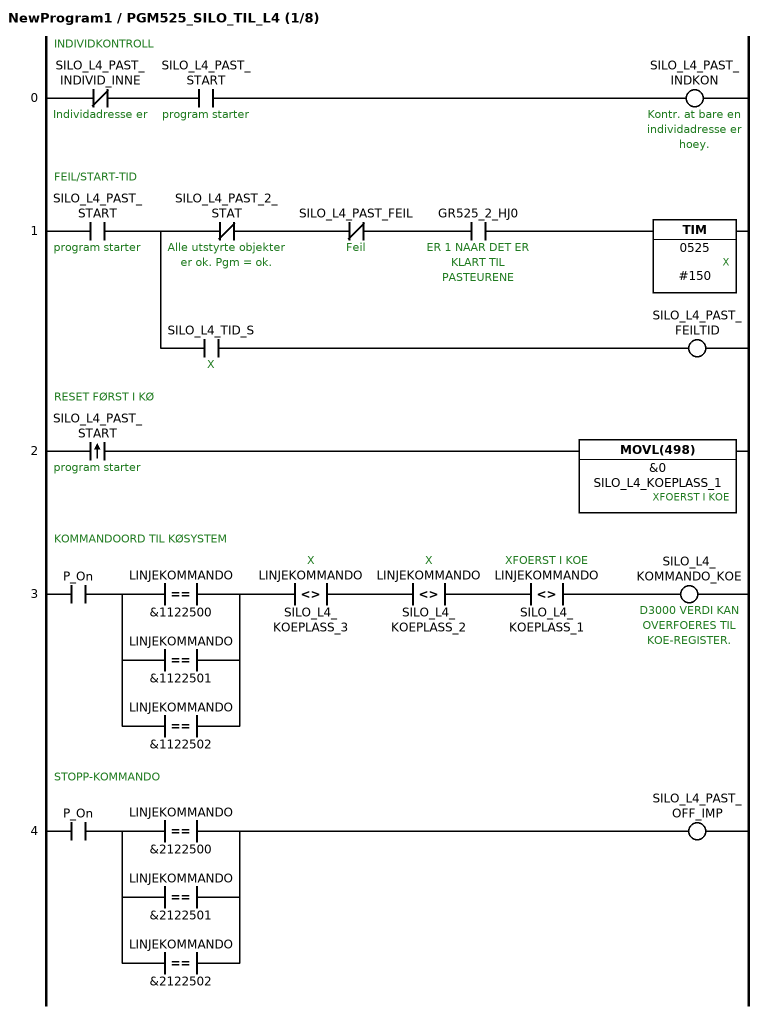
; [picture p672: NewProgram1 / PGM525_SILO_TIL_L4, rungs 0-4]
; rung 0: INDIVIDKONTROLL
LDNOT SILO_L4_PAST_INDIVID_INNE  ; Individadresse er
AND SILO_L4_PAST_START  ; program starter
OUT SILO_L4_PAST_INDKON  ; Kontr. at bare en individadresse er hoey.
; rung 1: FEIL/START-TID
LD SILO_L4_PAST_START  ; program starter
OUT TR0
ANDNOT SILO_L4_PAST_2_STAT  ; Alle utstyrte objekter er ok. Pgm = ok.
ANDNOT SILO_L4_PAST_FEIL  ; Feil
AND GR525_2_HJ0  ; ER 1 NAAR DET ER KLART TIL PASTEURENE
TIM 0525 #150  ; X
LD TR0
AND SILO_L4_TID_S  ; X
OUT SILO_L4_PAST_FEILTID
; rung 2: RESET FØRST I KØ
@LD SILO_L4_PAST_START  ; program starter
MOVL(498) &0 SILO_L4_KOEPLASS_1  ; XFOERST I KOE
; rung 3: KOMMANDOORD TIL KØSYSTEM
LD P_On
LD=L(301) LINJEKOMMANDO &1122500
OR=L(301) LINJEKOMMANDO &1122501
OR=L(301) LINJEKOMMANDO &1122502
ANDLD
AND<>L(306) LINJEKOMMANDO SILO_L4_KOEPLASS_3  ; X
AND<>L(306) LINJEKOMMANDO SILO_L4_KOEPLASS_2  ; X
AND<>L(306) LINJEKOMMANDO SILO_L4_KOEPLASS_1  ; XFOERST I KOE
OUT SILO_L4_KOMMANDO_KOE  ; D3000 VERDI KAN OVERFOERES TIL KOE-REGISTER.
; rung 4: STOPP-KOMMANDO
LD P_On
LD=L(301) LINJEKOMMANDO &2122500
OR=L(301) LINJEKOMMANDO &2122501
OR=L(301) LINJEKOMMANDO &2122502
ANDLD
OUT SILO_L4_PAST_OFF_IMP

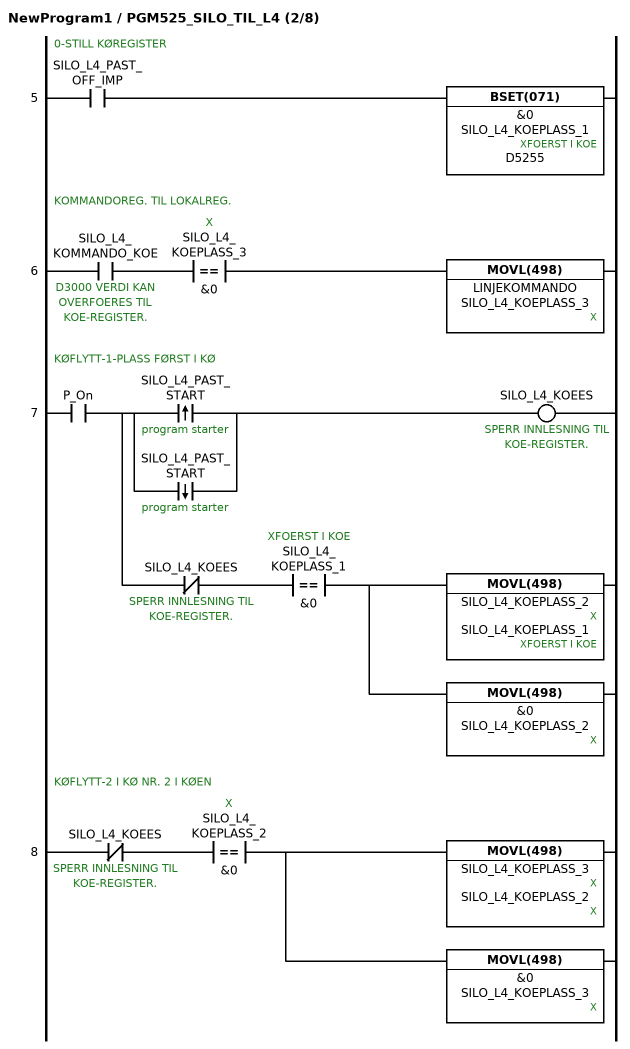
; rung 5: 0-STILL KØREGISTER
LD SILO_L4_PAST_OFF_IMP
BSET(071) &0 SILO_L4_KOEPLASS_1 D5255  ; XFOERST I KOE
; rung 6: KOMMANDOREG. TIL LOKALREG.
LD SILO_L4_KOMMANDO_KOE  ; D3000 VERDI KAN OVERFOERES TIL KOE-REGISTER.
AND=L(301) SILO_L4_KOEPLASS_3 &0  ; X
MOVL(498) LINJEKOMMANDO SILO_L4_KOEPLASS_3  ; X
; rung 7: KØFLYTT-1-PLASS FØRST I KØ
LD P_On
OUT TR0
@LD SILO_L4_PAST_START  ; program starter
%OR SILO_L4_PAST_START  ; program starter
ANDLD
OUT SILO_L4_KOEES  ; SPERR INNLESNING TIL KOE-REGISTER.
LD TR0
ANDNOT SILO_L4_KOEES  ; SPERR INNLESNING TIL KOE-REGISTER.
AND=L(301) SILO_L4_KOEPLASS_1 &0  ; XFOERST I KOE
MOVL(498) SILO_L4_KOEPLASS_2 SILO_L4_KOEPLASS_1  ; X, XFOERST I KOE
MOVL(498) &0 SILO_L4_KOEPLASS_2  ; X
; rung 8: KØFLYTT-2 I KØ NR. 2 I KØEN
LDNOT SILO_L4_KOEES  ; SPERR INNLESNING TIL KOE-REGISTER.
AND=L(301) SILO_L4_KOEPLASS_2 &0  ; X
MOVL(498) SILO_L4_KOEPLASS_3 SILO_L4_KOEPLASS_2  ; X
MOVL(498) &0 SILO_L4_KOEPLASS_3  ; X

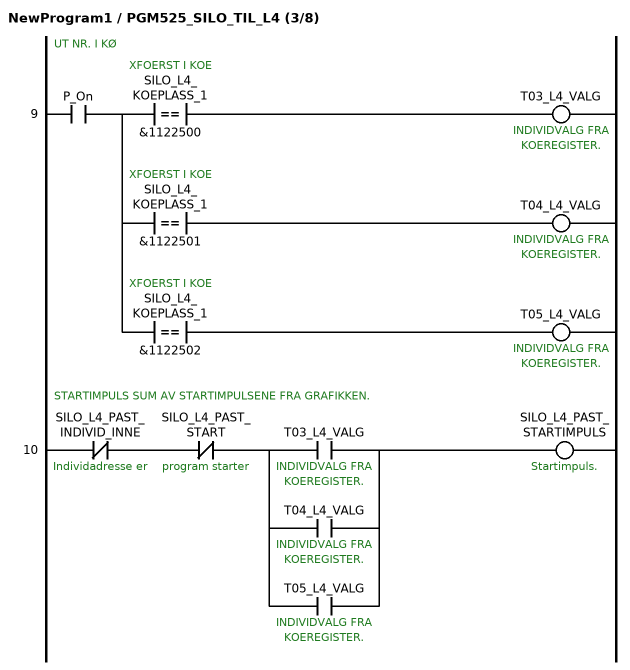
; rung 9: UT NR. I KØ
LD P_On
OUT TR0
AND=L(301) SILO_L4_KOEPLASS_1 &1122500  ; XFOERST I KOE
OUT T03_L4_VALG  ; INDIVIDVALG FRA KOEREGISTER.
LD TR0
AND=L(301) SILO_L4_KOEPLASS_1 &1122501  ; XFOERST I KOE
OUT T04_L4_VALG  ; INDIVIDVALG FRA KOEREGISTER.
LD TR0
AND=L(301) SILO_L4_KOEPLASS_1 &1122502  ; XFOERST I KOE
OUT T05_L4_VALG  ; INDIVIDVALG FRA KOEREGISTER.
; rung 10: STARTIMPULS SUM AV STARTIMPULSENE FRA GRAFIKKEN.
LDNOT SILO_L4_PAST_INDIVID_INNE  ; Individadresse er
ANDNOT SILO_L4_PAST_START  ; program starter
LD T03_L4_VALG  ; INDIVIDVALG FRA KOEREGISTER.
OR T04_L4_VALG  ; INDIVIDVALG FRA KOEREGISTER.
OR T05_L4_VALG  ; INDIVIDVALG FRA KOEREGISTER.
ANDLD
OUT SILO_L4_PAST_STARTIMPULS  ; Startimpuls.

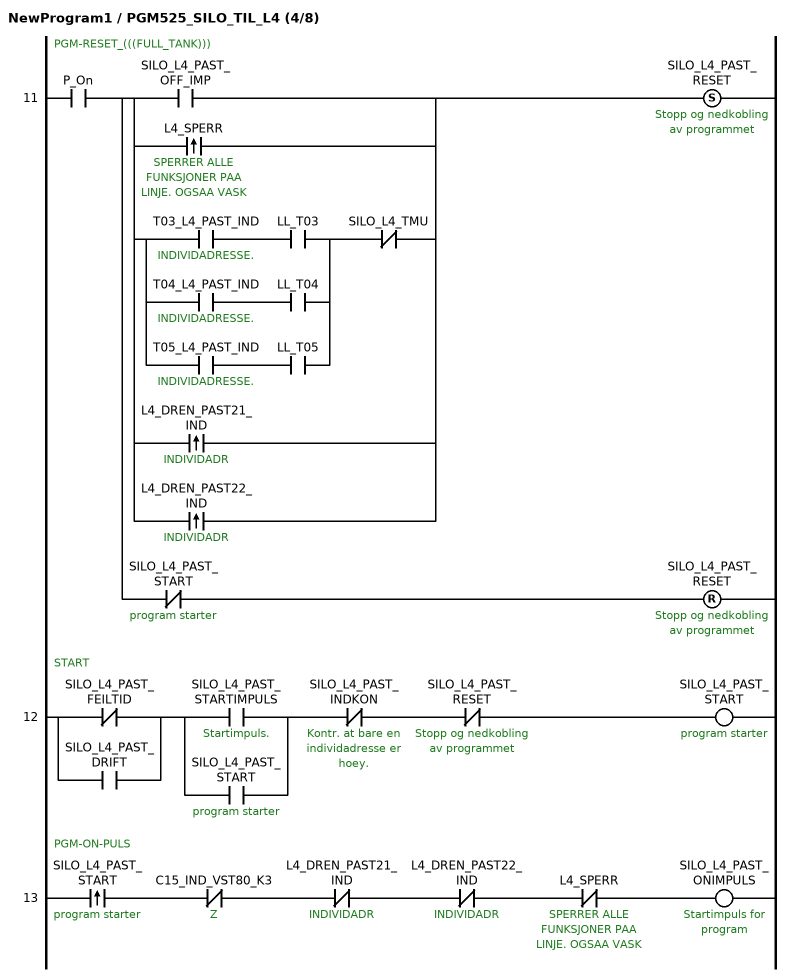
; rung 11: PGM-RESET_(((FULL_TANK)))
LD P_On
OUT TR0
LD SILO_L4_PAST_OFF_IMP
@OR L4_SPERR  ; SPERRER ALLE FUNKSJONER PAA LINJE. OGSAA VASK
LD T03_L4_PAST_IND  ; INDIVIDADRESSE.
AND LL_T03
LD T04_L4_PAST_IND  ; INDIVIDADRESSE.
AND LL_T04
ORLD
LD T05_L4_PAST_IND  ; INDIVIDADRESSE.
AND LL_T05
ORLD
ANDNOT SILO_L4_TMU
ORLD
@OR L4_DREN_PAST21_IND  ; INDIVIDADR
@OR L4_DREN_PAST22_IND  ; INDIVIDADR
ANDLD
SET SILO_L4_PAST_RESET  ; Stopp og nedkobling av programmet
LD TR0
ANDNOT SILO_L4_PAST_START  ; program starter
RSET SILO_L4_PAST_RESET  ; Stopp og nedkobling av programmet
; rung 12: START
LDNOT SILO_L4_PAST_FEILTID
OR SILO_L4_PAST_DRIFT
LD SILO_L4_PAST_STARTIMPULS  ; Startimpuls.
OR SILO_L4_PAST_START  ; program starter
ANDLD
ANDNOT SILO_L4_PAST_INDKON  ; Kontr. at bare en individadresse er hoey.
ANDNOT SILO_L4_PAST_RESET  ; Stopp og nedkobling av programmet
OUT SILO_L4_PAST_START  ; program starter
; rung 13: PGM-ON-PULS
@LD SILO_L4_PAST_START  ; program starter
ANDNOT C15_IND_VST80_K3  ; Z
ANDNOT L4_DREN_PAST21_IND  ; INDIVIDADR
ANDNOT L4_DREN_PAST22_IND  ; INDIVIDADR
ANDNOT L4_SPERR  ; SPERRER ALLE FUNKSJONER PAA LINJE. OGSAA VASK
OUT SILO_L4_PAST_ONIMPULS  ; Startimpuls for  program

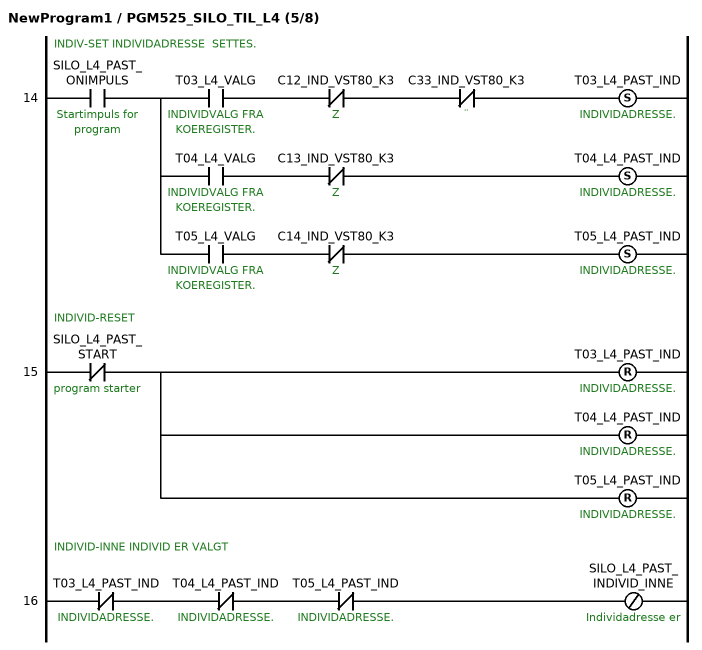
; rung 14: INDIV-SET INDIVIDADRESSE  SETTES.
LD SILO_L4_PAST_ONIMPULS  ; Startimpuls for  program
OUT TR0
AND T03_L4_VALG  ; INDIVIDVALG FRA KOEREGISTER.
ANDNOT C12_IND_VST80_K3  ; Z
ANDNOT C33_IND_VST80_K3  ; ¨
SET T03_L4_PAST_IND  ; INDIVIDADRESSE.
LD TR0
AND T04_L4_VALG  ; INDIVIDVALG FRA KOEREGISTER.
ANDNOT C13_IND_VST80_K3  ; Z
SET T04_L4_PAST_IND  ; INDIVIDADRESSE.
LD TR0
AND T05_L4_VALG  ; INDIVIDVALG FRA KOEREGISTER.
ANDNOT C14_IND_VST80_K3  ; Z
SET T05_L4_PAST_IND  ; INDIVIDADRESSE.
; rung 15: INDIVID-RESET
LDNOT SILO_L4_PAST_START  ; program starter
RSET T03_L4_PAST_IND  ; INDIVIDADRESSE.
RSET T04_L4_PAST_IND  ; INDIVIDADRESSE.
RSET T05_L4_PAST_IND  ; INDIVIDADRESSE.
; rung 16: INDIVID-INNE INDIVID ER VALGT
LDNOT T03_L4_PAST_IND  ; INDIVIDADRESSE.
ANDNOT T04_L4_PAST_IND  ; INDIVIDADRESSE.
ANDNOT T05_L4_PAST_IND  ; INDIVIDADRESSE.
OUTNOT SILO_L4_PAST_INDIVID_INNE  ; Individadresse er

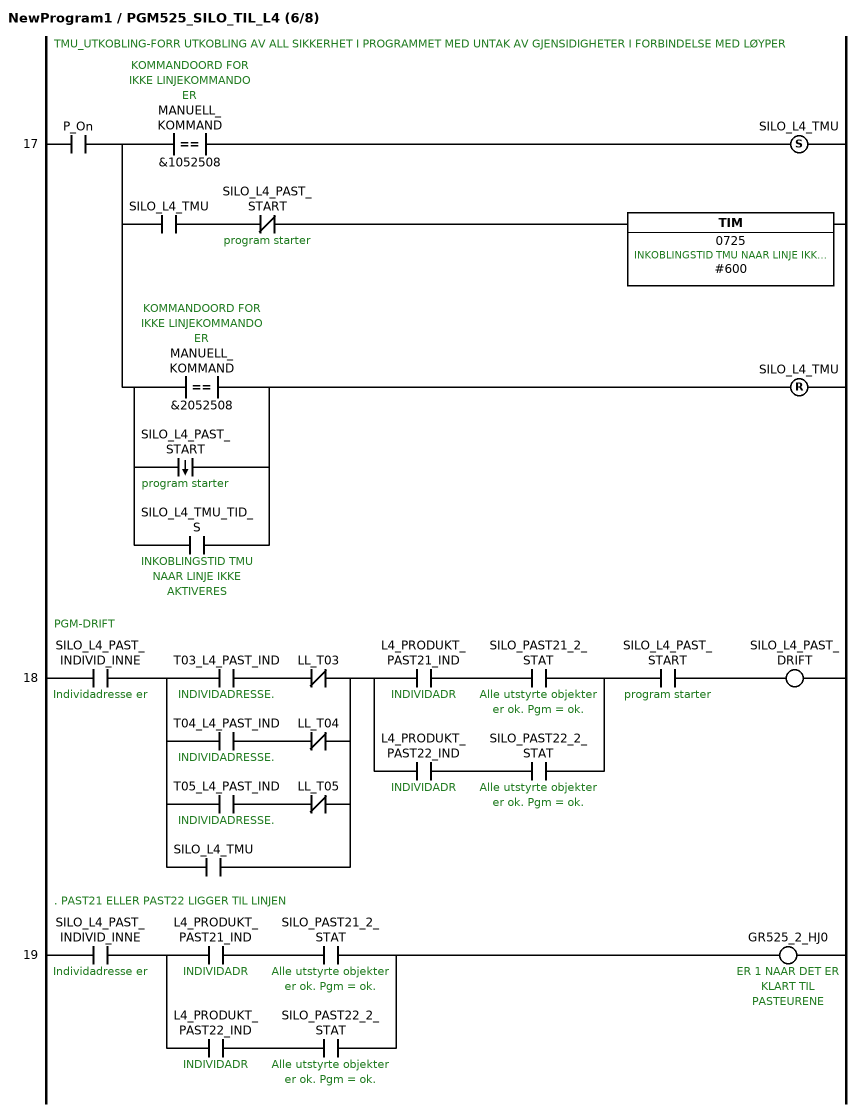
; rung 17: TMU_UTKOBLING-FORR UTKOBLING AV ALL SIKKERHET I PROGRAMMET MED UNTAK AV GJENSIDIGHETER I FORBINDELSE MED LØYPER
LD P_On
OUT TR0
AND=L(301) MANUELL_KOMMAND &1052508  ; KOMMANDOORD FOR IKKE LINJEKOMMANDOER
SET SILO_L4_TMU
LD TR0
AND SILO_L4_TMU
ANDNOT SILO_L4_PAST_START  ; program starter
TIM 0725 #600  ; INKOBLINGSTID TMU NAAR LINJE IKKE AKTIVERES
LD TR0
LD=L(301) MANUELL_KOMMAND &2052508  ; KOMMANDOORD FOR IKKE LINJEKOMMANDOER
%OR SILO_L4_PAST_START  ; program starter
OR SILO_L4_TMU_TID_S  ; INKOBLINGSTID TMU NAAR LINJE IKKE AKTIVERES
ANDLD
RSET SILO_L4_TMU
; rung 18: PGM-DRIFT
LD SILO_L4_PAST_INDIVID_INNE  ; Individadresse er
LD T03_L4_PAST_IND  ; INDIVIDADRESSE.
ANDNOT LL_T03
LD T04_L4_PAST_IND  ; INDIVIDADRESSE.
ANDNOT LL_T04
ORLD
LD T05_L4_PAST_IND  ; INDIVIDADRESSE.
ANDNOT LL_T05
ORLD
OR SILO_L4_TMU
ANDLD
LD L4_PRODUKT_PAST21_IND  ; INDIVIDADR
AND SILO_PAST21_2_STAT  ; Alle utstyrte objekter er ok. Pgm = ok.
LD L4_PRODUKT_PAST22_IND  ; INDIVIDADR
AND SILO_PAST22_2_STAT  ; Alle utstyrte objekter er ok. Pgm = ok.
ORLD
ANDLD
AND SILO_L4_PAST_START  ; program starter
OUT SILO_L4_PAST_DRIFT
; rung 19: . PAST21 ELLER PAST22 LIGGER TIL LINJEN
LD SILO_L4_PAST_INDIVID_INNE  ; Individadresse er
LD L4_PRODUKT_PAST21_IND  ; INDIVIDADR
AND SILO_PAST21_2_STAT  ; Alle utstyrte objekter er ok. Pgm = ok.
LD L4_PRODUKT_PAST22_IND  ; INDIVIDADR
AND SILO_PAST22_2_STAT  ; Alle utstyrte objekter er ok. Pgm = ok.
ORLD
ANDLD
OUT GR525_2_HJ0  ; ER 1 NAAR DET ER KLART TIL PASTEURENE

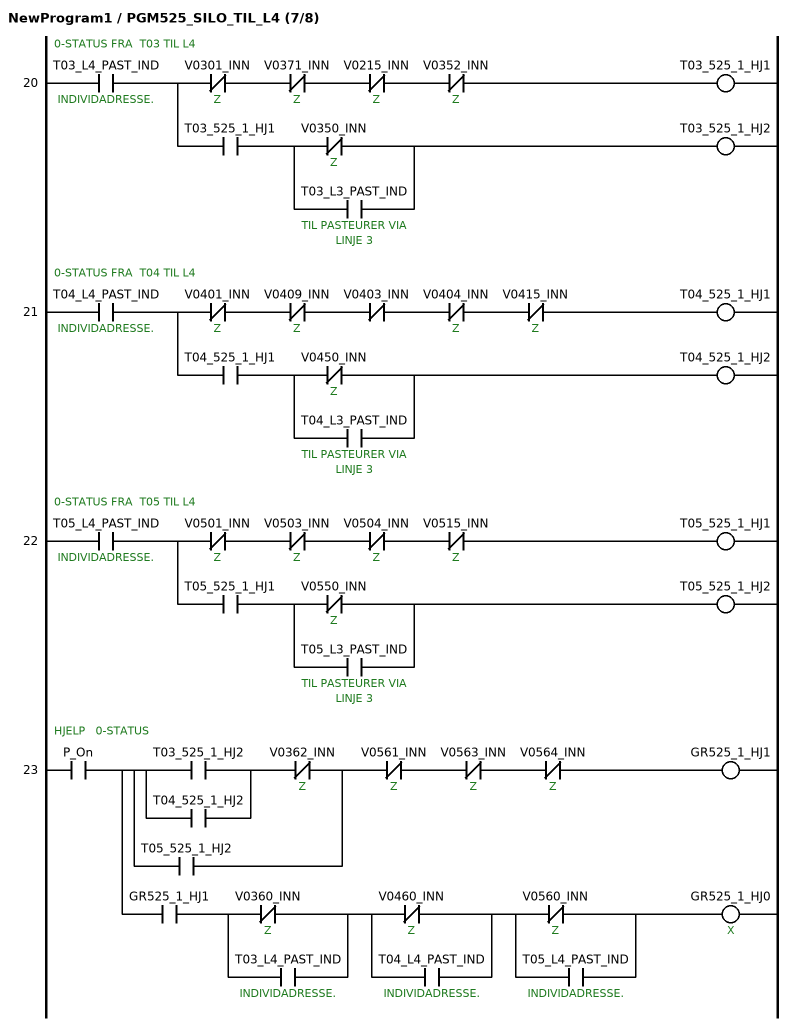
; rung 20: 0-STATUS FRA  T03 TIL L4
LD T03_L4_PAST_IND  ; INDIVIDADRESSE.
OUT TR0
ANDNOT V0301_INN  ; Z
ANDNOT V0371_INN  ; Z
ANDNOT V0215_INN  ; Z
ANDNOT V0352_INN  ; Z
OUT T03_525_1_HJ1
LD TR0
AND T03_525_1_HJ1
LDNOT V0350_INN  ; Z
OR T03_L3_PAST_IND  ; TIL PASTEURER VIA LINJE 3
ANDLD
OUT T03_525_1_HJ2
; rung 21: 0-STATUS FRA  T04 TIL L4
LD T04_L4_PAST_IND  ; INDIVIDADRESSE.
OUT TR0
ANDNOT V0401_INN  ; Z
ANDNOT V0409_INN  ; Z
ANDNOT V0403_INN
ANDNOT V0404_INN  ; Z
ANDNOT V0415_INN  ; Z
OUT T04_525_1_HJ1
LD TR0
AND T04_525_1_HJ1
LDNOT V0450_INN  ; Z
OR T04_L3_PAST_IND  ; TIL PASTEURER VIA LINJE 3
ANDLD
OUT T04_525_1_HJ2
; rung 22: 0-STATUS FRA  T05 TIL L4
LD T05_L4_PAST_IND  ; INDIVIDADRESSE.
OUT TR0
ANDNOT V0501_INN  ; Z
ANDNOT V0503_INN  ; Z
ANDNOT V0504_INN  ; Z
ANDNOT V0515_INN  ; Z
OUT T05_525_1_HJ1
LD TR0
AND T05_525_1_HJ1
LDNOT V0550_INN  ; Z
OR T05_L3_PAST_IND  ; TIL PASTEURER VIA LINJE 3
ANDLD
OUT T05_525_1_HJ2
; rung 23: HJELP   0-STATUS
LD P_On
OUT TR0
LD T03_525_1_HJ2
OR T04_525_1_HJ2
ANDNOT V0362_INN  ; Z
OR T05_525_1_HJ2
ANDLD
ANDNOT V0561_INN  ; Z
ANDNOT V0563_INN  ; Z
ANDNOT V0564_INN  ; Z
OUT GR525_1_HJ1
LD TR0
AND GR525_1_HJ1
LDNOT V0360_INN  ; Z
OR T03_L4_PAST_IND  ; INDIVIDADRESSE.
ANDLD
LDNOT V0460_INN  ; Z
OR T04_L4_PAST_IND  ; INDIVIDADRESSE.
ANDLD
LDNOT V0560_INN  ; Z
OR T05_L4_PAST_IND  ; INDIVIDADRESSE.
ANDLD
OUT GR525_1_HJ0  ; X

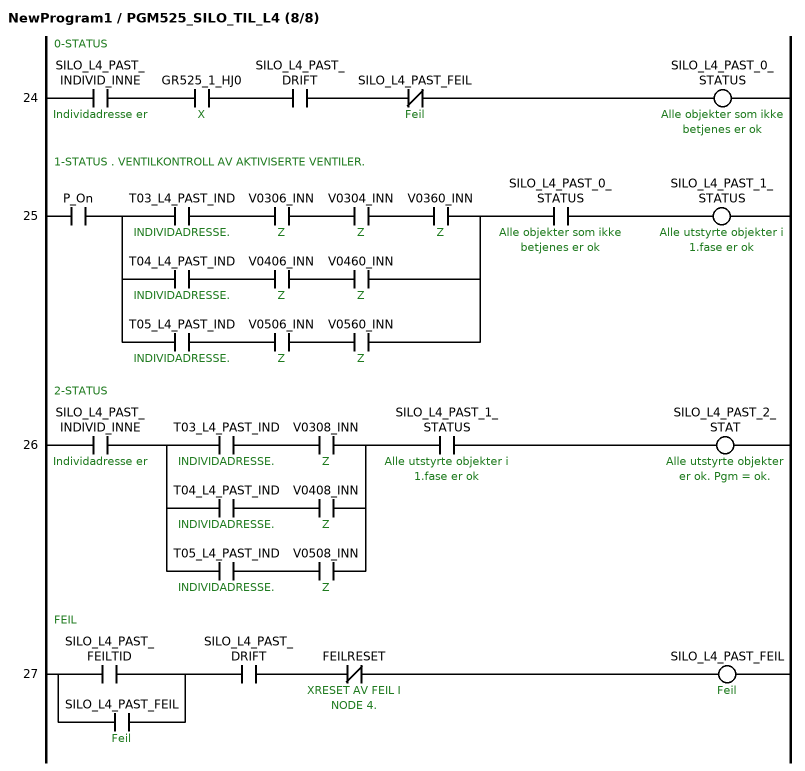
; rung 24: 0-STATUS
LD SILO_L4_PAST_INDIVID_INNE  ; Individadresse er
AND GR525_1_HJ0  ; X
AND SILO_L4_PAST_DRIFT
ANDNOT SILO_L4_PAST_FEIL  ; Feil
OUT SILO_L4_PAST_0_STATUS  ; Alle objekter som ikke betjenes er ok
; rung 25: 1-STATUS . VENTILKONTROLL AV AKTIVISERTE VENTILER.
LD P_On
LD T03_L4_PAST_IND  ; INDIVIDADRESSE.
AND V0306_INN  ; Z
AND V0304_INN  ; Z
AND V0360_INN  ; Z
LD T04_L4_PAST_IND  ; INDIVIDADRESSE.
AND V0406_INN  ; Z
AND V0460_INN  ; Z
ORLD
LD T05_L4_PAST_IND  ; INDIVIDADRESSE.
AND V0506_INN  ; Z
AND V0560_INN  ; Z
ORLD
ANDLD
AND SILO_L4_PAST_0_STATUS  ; Alle objekter som ikke betjenes er ok
OUT SILO_L4_PAST_1_STATUS  ; Alle utstyrte objekter i 1.fase er ok
; rung 26: 2-STATUS
LD SILO_L4_PAST_INDIVID_INNE  ; Individadresse er
LD T03_L4_PAST_IND  ; INDIVIDADRESSE.
AND V0308_INN  ; Z
LD T04_L4_PAST_IND  ; INDIVIDADRESSE.
AND V0408_INN  ; Z
ORLD
LD T05_L4_PAST_IND  ; INDIVIDADRESSE.
AND V0508_INN  ; Z
ORLD
ANDLD
AND SILO_L4_PAST_1_STATUS  ; Alle utstyrte objekter i 1.fase er ok
OUT SILO_L4_PAST_2_STAT  ; Alle utstyrte objekter er ok. Pgm = ok.
; rung 27: FEIL
LD SILO_L4_PAST_FEILTID
OR SILO_L4_PAST_FEIL  ; Feil
AND SILO_L4_PAST_DRIFT
ANDNOT FEILRESET  ; XRESET AV FEIL I NODE 4.
OUT SILO_L4_PAST_FEIL  ; Feil

### Section PGM526_TIL_PAST21

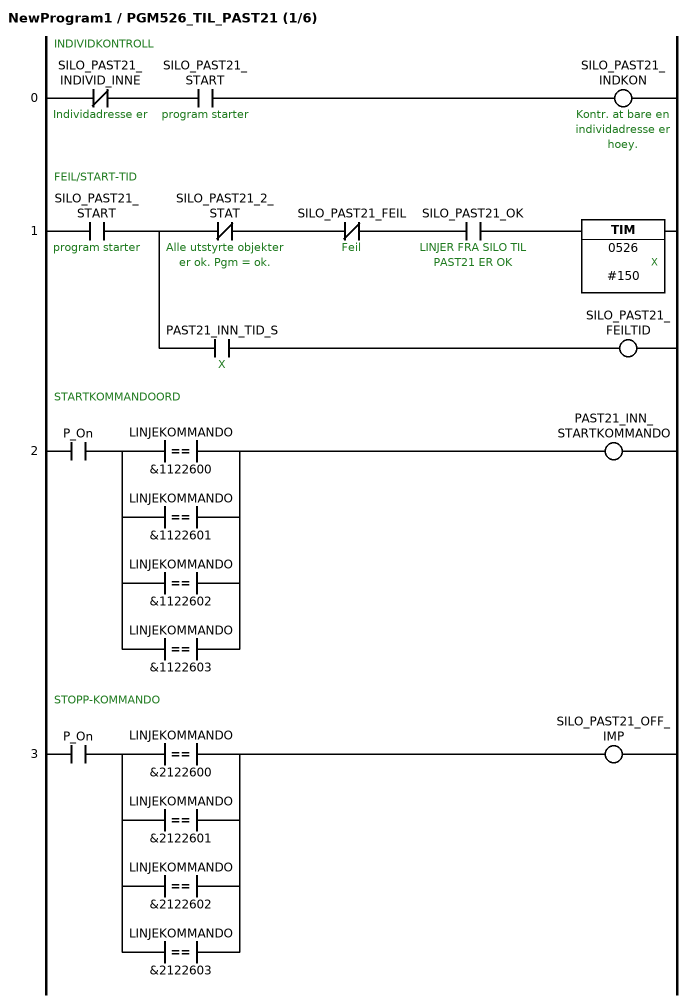
; rung 0: INDIVIDKONTROLL
LDNOT SILO_PAST21_INDIVID_INNE  ; Individadresse er
AND SILO_PAST21_START  ; program starter
OUT SILO_PAST21_INDKON  ; Kontr. at bare en individadresse er hoey.
; rung 1: FEIL/START-TID
LD SILO_PAST21_START  ; program starter
OUT TR0
ANDNOT SILO_PAST21_2_STAT  ; Alle utstyrte objekter er ok. Pgm = ok.
ANDNOT SILO_PAST21_FEIL  ; Feil
AND SILO_PAST21_OK  ; LINJER FRA SILO TIL  PAST21 ER OK
TIM 0526 #150  ; X
LD TR0
AND PAST21_INN_TID_S  ; X
OUT SILO_PAST21_FEILTID
; rung 2: STARTKOMMANDOORD
LD P_On
LD=L(301) LINJEKOMMANDO &1122600
OR=L(301) LINJEKOMMANDO &1122601
OR=L(301) LINJEKOMMANDO &1122602
OR=L(301) LINJEKOMMANDO &1122603
ANDLD
OUT PAST21_INN_STARTKOMMANDO
; rung 3: STOPP-KOMMANDO
LD P_On
LD=L(301) LINJEKOMMANDO &2122600
OR=L(301) LINJEKOMMANDO &2122601
OR=L(301) LINJEKOMMANDO &2122602
OR=L(301) LINJEKOMMANDO &2122603
ANDLD
OUT SILO_PAST21_OFF_IMP

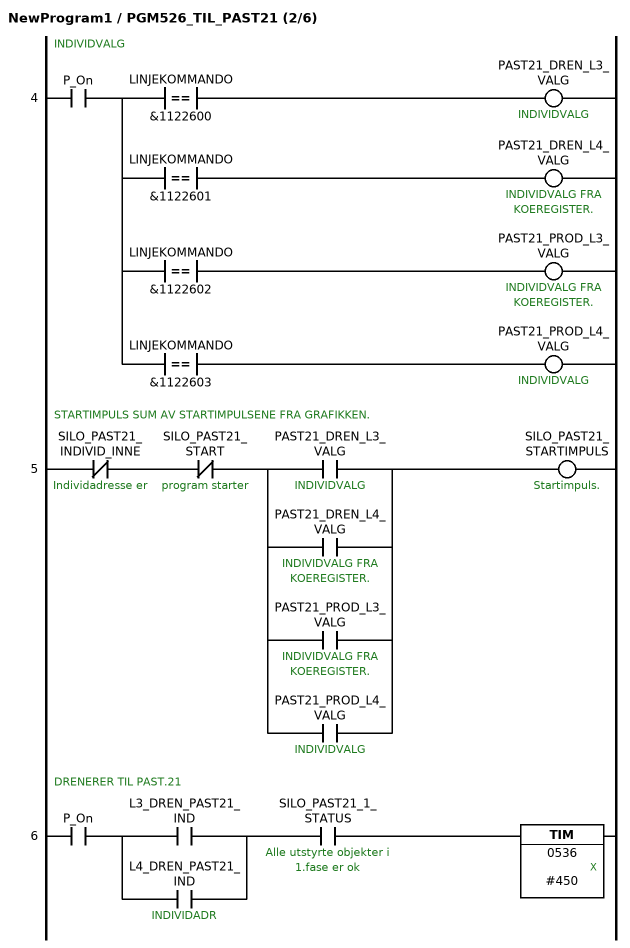
; rung 4: INDIVIDVALG
LD P_On
OUT TR0
AND=L(301) LINJEKOMMANDO &1122600
OUT PAST21_DREN_L3_VALG  ; INDIVIDVALG
LD TR0
AND=L(301) LINJEKOMMANDO &1122601
OUT PAST21_DREN_L4_VALG  ; INDIVIDVALG FRA KOEREGISTER.
LD TR0
AND=L(301) LINJEKOMMANDO &1122602
OUT PAST21_PROD_L3_VALG  ; INDIVIDVALG FRA KOEREGISTER.
LD TR0
AND=L(301) LINJEKOMMANDO &1122603
OUT PAST21_PROD_L4_VALG  ; INDIVIDVALG
; rung 5: STARTIMPULS SUM AV STARTIMPULSENE FRA GRAFIKKEN.
LDNOT SILO_PAST21_INDIVID_INNE  ; Individadresse er
ANDNOT SILO_PAST21_START  ; program starter
LD PAST21_DREN_L3_VALG  ; INDIVIDVALG
OR PAST21_DREN_L4_VALG  ; INDIVIDVALG FRA KOEREGISTER.
OR PAST21_PROD_L3_VALG  ; INDIVIDVALG FRA KOEREGISTER.
OR PAST21_PROD_L4_VALG  ; INDIVIDVALG
ANDLD
OUT SILO_PAST21_STARTIMPULS  ; Startimpuls.
; rung 6: DRENERER TIL PAST.21
LD P_On
LD L3_DREN_PAST21_IND
OR L4_DREN_PAST21_IND  ; INDIVIDADR
ANDLD
AND SILO_PAST21_1_STATUS  ; Alle utstyrte objekter i 1.fase er ok
TIM 0536 #450  ; X

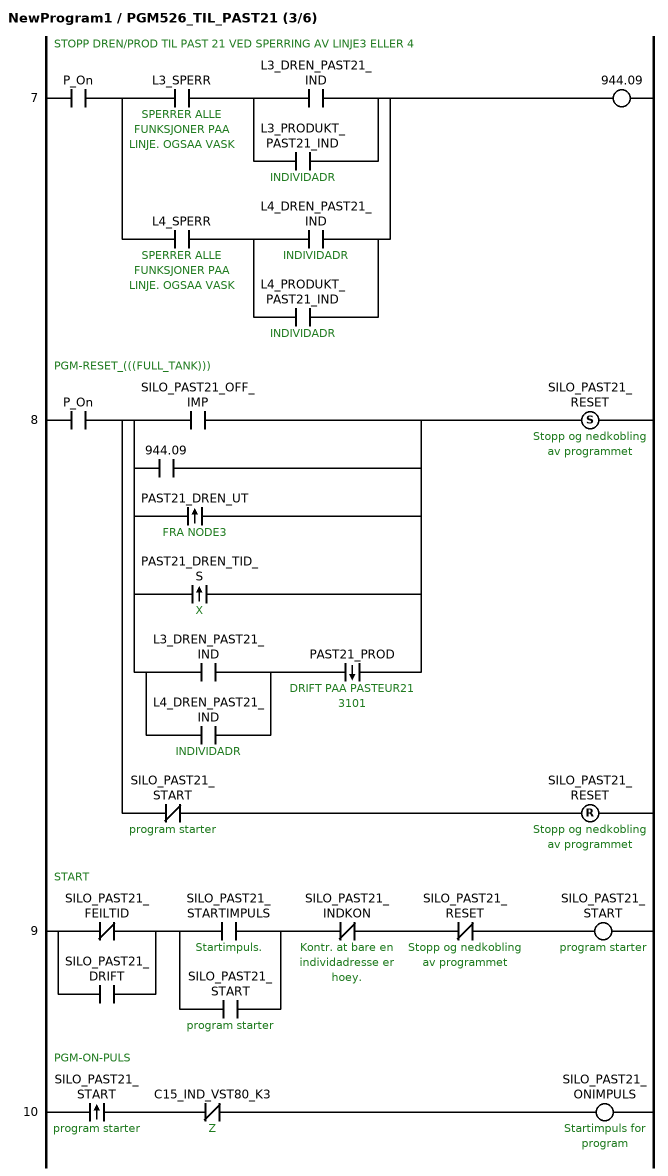
; rung 7: STOPP DREN/PROD TIL PAST 21 VED SPERRING AV LINJE3 ELLER 4
LD P_On
LD L3_SPERR  ; SPERRER ALLE FUNKSJONER PAA LINJE. OGSAA VASK
LD L3_DREN_PAST21_IND
OR L3_PRODUKT_PAST21_IND  ; INDIVIDADR
ANDLD
LD L4_SPERR  ; SPERRER ALLE FUNKSJONER PAA LINJE. OGSAA VASK
LD L4_DREN_PAST21_IND  ; INDIVIDADR
OR L4_PRODUKT_PAST21_IND  ; INDIVIDADR
ANDLD
ORLD
ANDLD
OUT 944.09
; rung 8: PGM-RESET_(((FULL_TANK)))
LD P_On
OUT TR0
LD SILO_PAST21_OFF_IMP
OR 944.09
@OR PAST21_DREN_UT  ; FRA NODE3
@OR PAST21_DREN_TID_S  ; X
LD L3_DREN_PAST21_IND
OR L4_DREN_PAST21_IND  ; INDIVIDADR
%AND PAST21_PROD  ; DRIFT PAA PASTEUR21 3101
ORLD
ANDLD
SET SILO_PAST21_RESET  ; Stopp og nedkobling av programmet
LD TR0
ANDNOT SILO_PAST21_START  ; program starter
RSET SILO_PAST21_RESET  ; Stopp og nedkobling av programmet
; rung 9: START
LDNOT SILO_PAST21_FEILTID
OR SILO_PAST21_DRIFT
LD SILO_PAST21_STARTIMPULS  ; Startimpuls.
OR SILO_PAST21_START  ; program starter
ANDLD
ANDNOT SILO_PAST21_INDKON  ; Kontr. at bare en individadresse er hoey.
ANDNOT SILO_PAST21_RESET  ; Stopp og nedkobling av programmet
OUT SILO_PAST21_START  ; program starter
; rung 10: PGM-ON-PULS
@LD SILO_PAST21_START  ; program starter
ANDNOT C15_IND_VST80_K3  ; Z
OUT SILO_PAST21_ONIMPULS  ; Startimpuls for  program

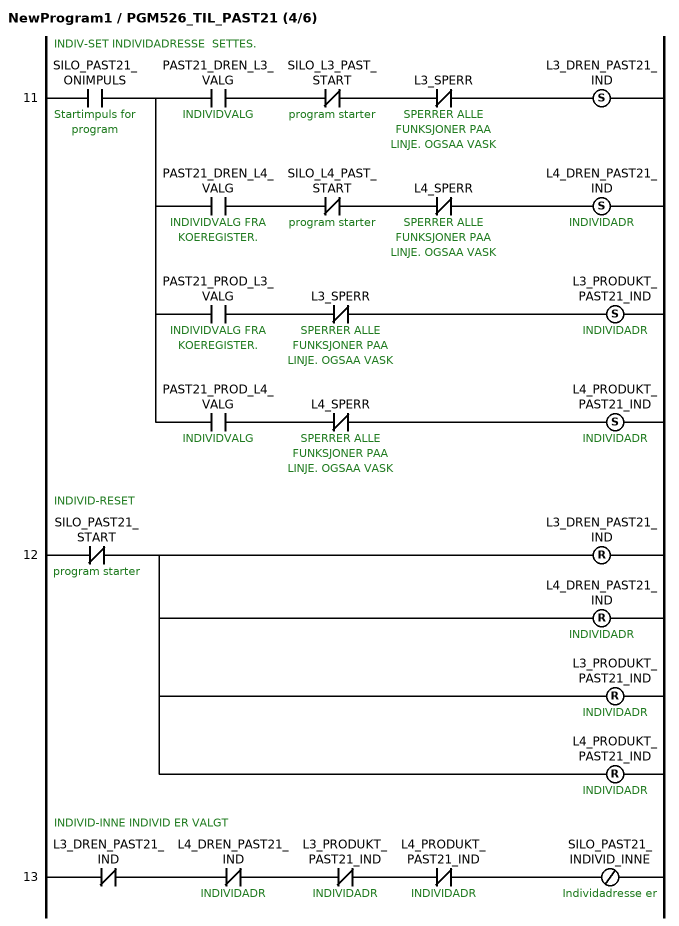
; rung 11: INDIV-SET INDIVIDADRESSE  SETTES.
LD SILO_PAST21_ONIMPULS  ; Startimpuls for  program
OUT TR0
AND PAST21_DREN_L3_VALG  ; INDIVIDVALG
ANDNOT SILO_L3_PAST_START  ; program starter
ANDNOT L3_SPERR  ; SPERRER ALLE FUNKSJONER PAA LINJE. OGSAA VASK
SET L3_DREN_PAST21_IND
LD TR0
AND PAST21_DREN_L4_VALG  ; INDIVIDVALG FRA KOEREGISTER.
ANDNOT SILO_L4_PAST_START  ; program starter
ANDNOT L4_SPERR  ; SPERRER ALLE FUNKSJONER PAA LINJE. OGSAA VASK
SET L4_DREN_PAST21_IND  ; INDIVIDADR
LD TR0
AND PAST21_PROD_L3_VALG  ; INDIVIDVALG FRA KOEREGISTER.
ANDNOT L3_SPERR  ; SPERRER ALLE FUNKSJONER PAA LINJE. OGSAA VASK
SET L3_PRODUKT_PAST21_IND  ; INDIVIDADR
LD TR0
AND PAST21_PROD_L4_VALG  ; INDIVIDVALG
ANDNOT L4_SPERR  ; SPERRER ALLE FUNKSJONER PAA LINJE. OGSAA VASK
SET L4_PRODUKT_PAST21_IND  ; INDIVIDADR
; rung 12: INDIVID-RESET
LDNOT SILO_PAST21_START  ; program starter
RSET L3_DREN_PAST21_IND
RSET L4_DREN_PAST21_IND  ; INDIVIDADR
RSET L3_PRODUKT_PAST21_IND  ; INDIVIDADR
RSET L4_PRODUKT_PAST21_IND  ; INDIVIDADR
; rung 13: INDIVID-INNE INDIVID ER VALGT
LDNOT L3_DREN_PAST21_IND
ANDNOT L4_DREN_PAST21_IND  ; INDIVIDADR
ANDNOT L3_PRODUKT_PAST21_IND  ; INDIVIDADR
ANDNOT L4_PRODUKT_PAST21_IND  ; INDIVIDADR
OUTNOT SILO_PAST21_INDIVID_INNE  ; Individadresse er

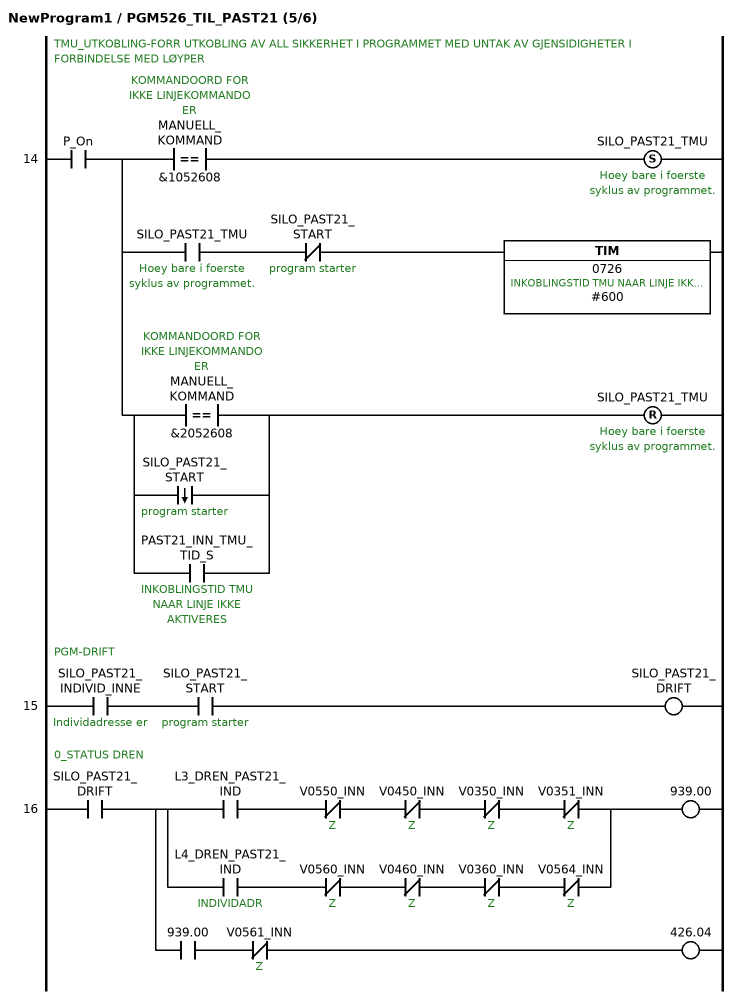
; rung 14: TMU_UTKOBLING-FORR UTKOBLING AV ALL SIKKERHET I PROGRAMMET MED UNTAK AV GJENSIDIGHETER I FORBINDELSE MED LØYPER
LD P_On
OUT TR0
AND=L(301) MANUELL_KOMMAND &1052608  ; KOMMANDOORD FOR IKKE LINJEKOMMANDOER
SET SILO_PAST21_TMU  ; Hoey bare i foerste syklus av programmet.
LD TR0
AND SILO_PAST21_TMU  ; Hoey bare i foerste syklus av programmet.
ANDNOT SILO_PAST21_START  ; program starter
TIM 0726 #600  ; INKOBLINGSTID TMU NAAR LINJE IKKE AKTIVERES
LD TR0
LD=L(301) MANUELL_KOMMAND &2052608  ; KOMMANDOORD FOR IKKE LINJEKOMMANDOER
%OR SILO_PAST21_START  ; program starter
OR PAST21_INN_TMU_TID_S  ; INKOBLINGSTID TMU NAAR LINJE IKKE AKTIVERES
ANDLD
RSET SILO_PAST21_TMU  ; Hoey bare i foerste syklus av programmet.
; rung 15: PGM-DRIFT
LD SILO_PAST21_INDIVID_INNE  ; Individadresse er
AND SILO_PAST21_START  ; program starter
OUT SILO_PAST21_DRIFT
; rung 16: 0_STATUS DREN
LD SILO_PAST21_DRIFT
OUT TR0
LD L3_DREN_PAST21_IND
ANDNOT V0550_INN  ; Z
ANDNOT V0450_INN  ; Z
ANDNOT V0350_INN  ; Z
ANDNOT V0351_INN  ; Z
LD L4_DREN_PAST21_IND  ; INDIVIDADR
ANDNOT V0560_INN  ; Z
ANDNOT V0460_INN  ; Z
ANDNOT V0360_INN  ; Z
ANDNOT V0564_INN  ; Z
ORLD
ANDLD
OUT 939.00
LD TR0
AND 939.00
ANDNOT V0561_INN  ; Z
OUT 426.04

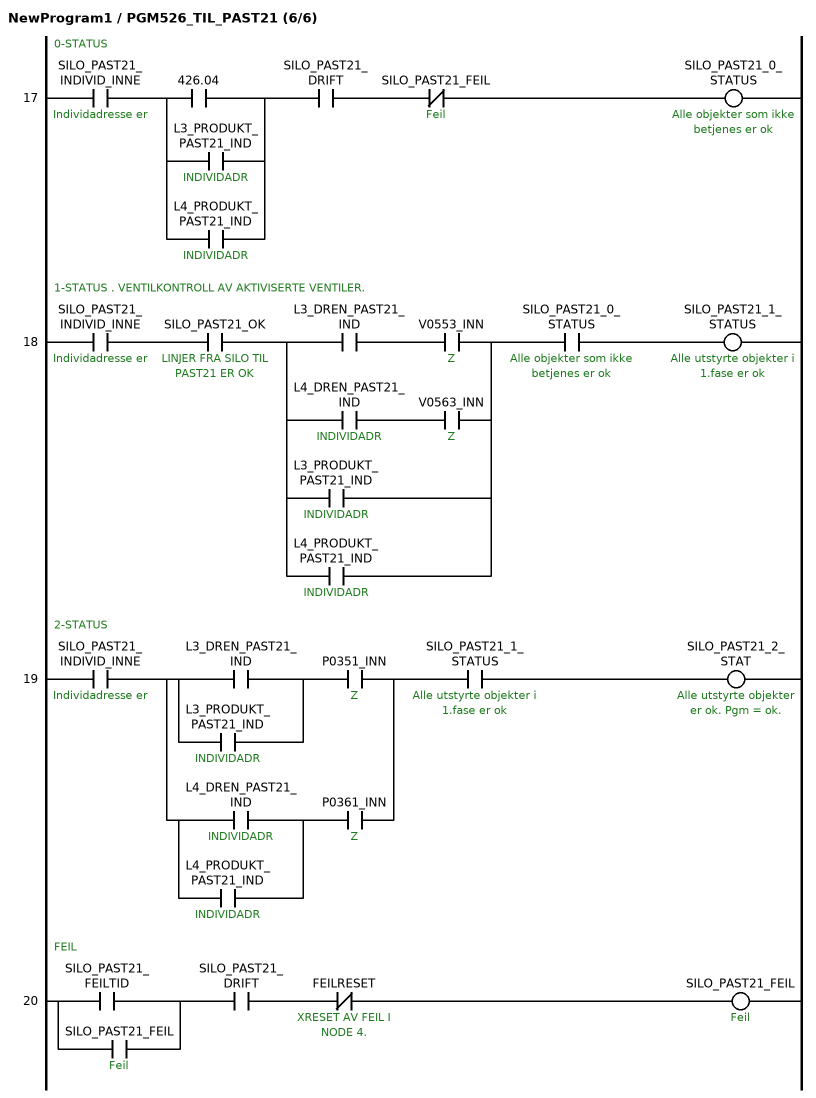
; rung 17: 0-STATUS
LD SILO_PAST21_INDIVID_INNE  ; Individadresse er
LD 426.04
OR L3_PRODUKT_PAST21_IND  ; INDIVIDADR
OR L4_PRODUKT_PAST21_IND  ; INDIVIDADR
ANDLD
AND SILO_PAST21_DRIFT
ANDNOT SILO_PAST21_FEIL  ; Feil
OUT SILO_PAST21_0_STATUS  ; Alle objekter som ikke betjenes er ok
; rung 18: 1-STATUS . VENTILKONTROLL AV AKTIVISERTE VENTILER.
LD SILO_PAST21_INDIVID_INNE  ; Individadresse er
AND SILO_PAST21_OK  ; LINJER FRA SILO TIL  PAST21 ER OK
LD L3_DREN_PAST21_IND
AND V0553_INN  ; Z
LD L4_DREN_PAST21_IND  ; INDIVIDADR
AND V0563_INN  ; Z
ORLD
OR L3_PRODUKT_PAST21_IND  ; INDIVIDADR
OR L4_PRODUKT_PAST21_IND  ; INDIVIDADR
ANDLD
AND SILO_PAST21_0_STATUS  ; Alle objekter som ikke betjenes er ok
OUT SILO_PAST21_1_STATUS  ; Alle utstyrte objekter i 1.fase er ok
; rung 19: 2-STATUS
LD SILO_PAST21_INDIVID_INNE  ; Individadresse er
LD L3_DREN_PAST21_IND
OR L3_PRODUKT_PAST21_IND  ; INDIVIDADR
AND P0351_INN  ; Z
LD L4_DREN_PAST21_IND  ; INDIVIDADR
OR L4_PRODUKT_PAST21_IND  ; INDIVIDADR
AND P0361_INN  ; Z
ORLD
ANDLD
AND SILO_PAST21_1_STATUS  ; Alle utstyrte objekter i 1.fase er ok
OUT SILO_PAST21_2_STAT  ; Alle utstyrte objekter er ok. Pgm = ok.
; rung 20: FEIL
LD SILO_PAST21_FEILTID
OR SILO_PAST21_FEIL  ; Feil
AND SILO_PAST21_DRIFT
ANDNOT FEILRESET  ; XRESET AV FEIL I NODE 4.
OUT SILO_PAST21_FEIL  ; Feil

### Section L3_STATUS

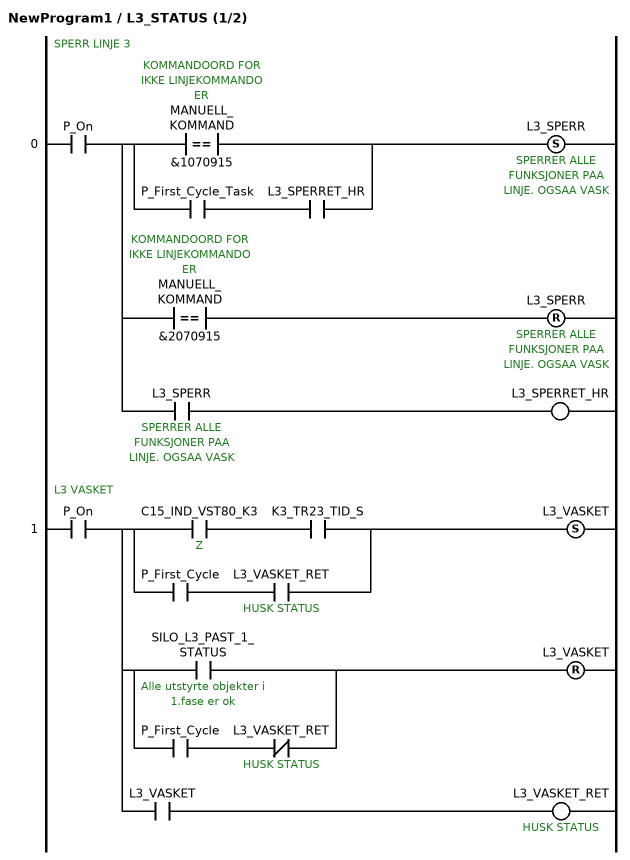
; rung 0: SPERR LINJE 3
LD P_On
OUT TR0
LD=L(301) MANUELL_KOMMAND &1070915  ; KOMMANDOORD FOR IKKE LINJEKOMMANDOER
LD P_First_Cycle_Task
AND L3_SPERRET_HR
ORLD
ANDLD
SET L3_SPERR  ; SPERRER ALLE FUNKSJONER PAA LINJE. OGSAA VASK
LD TR0
AND=L(301) MANUELL_KOMMAND &2070915  ; KOMMANDOORD FOR IKKE LINJEKOMMANDOER
RSET L3_SPERR  ; SPERRER ALLE FUNKSJONER PAA LINJE. OGSAA VASK
LD TR0
AND L3_SPERR  ; SPERRER ALLE FUNKSJONER PAA LINJE. OGSAA VASK
OUT L3_SPERRET_HR
; rung 1: L3 VASKET
LD P_On
OUT TR0
LD C15_IND_VST80_K3  ; Z
AND K3_TR23_TID_S
LD P_First_Cycle
AND L3_VASKET_RET  ; HUSK STATUS
ORLD
ANDLD
SET L3_VASKET
LD TR0
LD SILO_L3_PAST_1_STATUS  ; Alle utstyrte objekter i 1.fase er ok
LD P_First_Cycle
ANDNOT L3_VASKET_RET  ; HUSK STATUS
ORLD
ANDLD
RSET L3_VASKET
LD TR0
AND L3_VASKET
OUT L3_VASKET_RET  ; HUSK STATUS

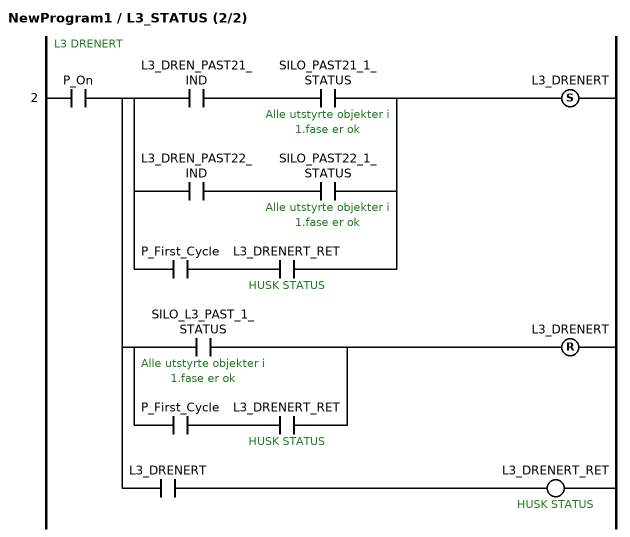
; rung 2: L3 DRENERT
LD P_On
OUT TR0
LD L3_DREN_PAST21_IND
AND SILO_PAST21_1_STATUS  ; Alle utstyrte objekter i 1.fase er ok
LD L3_DREN_PAST22_IND
AND SILO_PAST22_1_STATUS  ; Alle utstyrte objekter i 1.fase er ok
ORLD
LD P_First_Cycle
AND L3_DRENERT_RET  ; HUSK STATUS
ORLD
ANDLD
SET L3_DRENERT
LD TR0
LD SILO_L3_PAST_1_STATUS  ; Alle utstyrte objekter i 1.fase er ok
LD P_First_Cycle
AND L3_DRENERT_RET  ; HUSK STATUS
ORLD
ANDLD
RSET L3_DRENERT
LD TR0
AND L3_DRENERT
OUT L3_DRENERT_RET  ; HUSK STATUS

### Section PGM527_TIL_PAST22

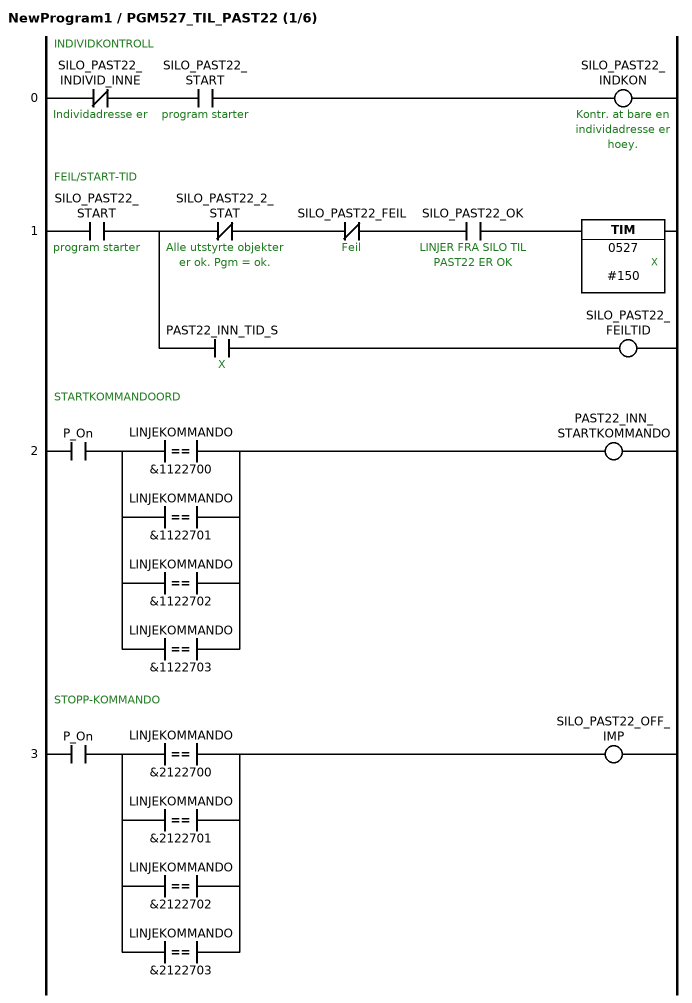
; rung 0: INDIVIDKONTROLL
LDNOT SILO_PAST22_INDIVID_INNE  ; Individadresse er
AND SILO_PAST22_START  ; program starter
OUT SILO_PAST22_INDKON  ; Kontr. at bare en individadresse er hoey.
; rung 1: FEIL/START-TID
LD SILO_PAST22_START  ; program starter
OUT TR0
ANDNOT SILO_PAST22_2_STAT  ; Alle utstyrte objekter er ok. Pgm = ok.
ANDNOT SILO_PAST22_FEIL  ; Feil
AND SILO_PAST22_OK  ; LINJER FRA SILO TIL  PAST22 ER OK
TIM 0527 #150  ; X
LD TR0
AND PAST22_INN_TID_S  ; X
OUT SILO_PAST22_FEILTID
; rung 2: STARTKOMMANDOORD
LD P_On
LD=L(301) LINJEKOMMANDO &1122700
OR=L(301) LINJEKOMMANDO &1122701
OR=L(301) LINJEKOMMANDO &1122702
OR=L(301) LINJEKOMMANDO &1122703
ANDLD
OUT PAST22_INN_STARTKOMMANDO
; rung 3: STOPP-KOMMANDO
LD P_On
LD=L(301) LINJEKOMMANDO &2122700
OR=L(301) LINJEKOMMANDO &2122701
OR=L(301) LINJEKOMMANDO &2122702
OR=L(301) LINJEKOMMANDO &2122703
ANDLD
OUT SILO_PAST22_OFF_IMP

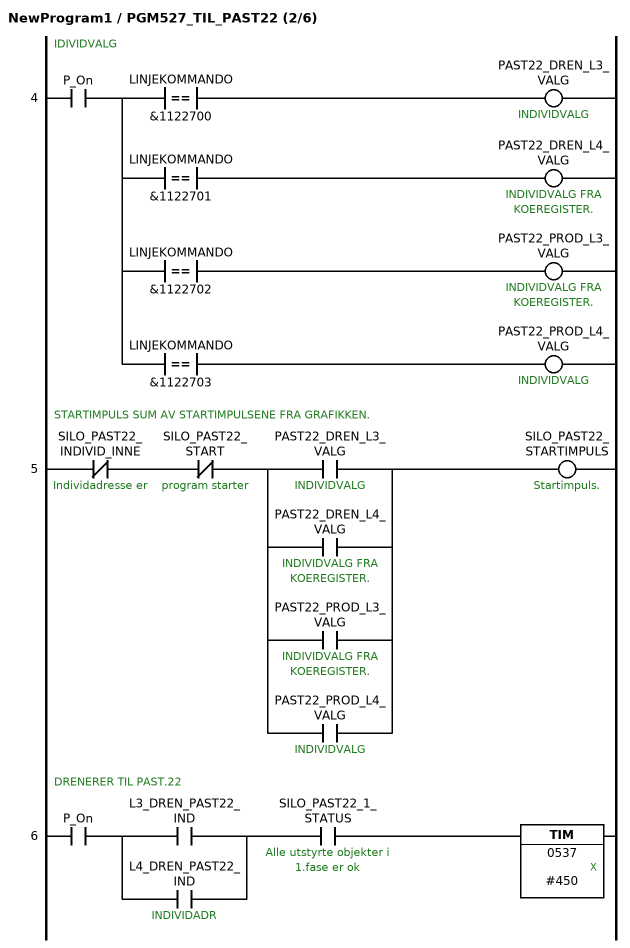
; rung 4: IDIVIDVALG
LD P_On
OUT TR0
AND=L(301) LINJEKOMMANDO &1122700
OUT PAST22_DREN_L3_VALG  ; INDIVIDVALG
LD TR0
AND=L(301) LINJEKOMMANDO &1122701
OUT PAST22_DREN_L4_VALG  ; INDIVIDVALG FRA KOEREGISTER.
LD TR0
AND=L(301) LINJEKOMMANDO &1122702
OUT PAST22_PROD_L3_VALG  ; INDIVIDVALG FRA KOEREGISTER.
LD TR0
AND=L(301) LINJEKOMMANDO &1122703
OUT PAST22_PROD_L4_VALG  ; INDIVIDVALG
; rung 5: STARTIMPULS SUM AV STARTIMPULSENE FRA GRAFIKKEN.
LDNOT SILO_PAST22_INDIVID_INNE  ; Individadresse er
ANDNOT SILO_PAST22_START  ; program starter
LD PAST22_DREN_L3_VALG  ; INDIVIDVALG
OR PAST22_DREN_L4_VALG  ; INDIVIDVALG FRA KOEREGISTER.
OR PAST22_PROD_L3_VALG  ; INDIVIDVALG FRA KOEREGISTER.
OR PAST22_PROD_L4_VALG  ; INDIVIDVALG
ANDLD
OUT SILO_PAST22_STARTIMPULS  ; Startimpuls.
; rung 6: DRENERER TIL PAST.22
LD P_On
LD L3_DREN_PAST22_IND
OR L4_DREN_PAST22_IND  ; INDIVIDADR
ANDLD
AND SILO_PAST22_1_STATUS  ; Alle utstyrte objekter i 1.fase er ok
TIM 0537 #450  ; X

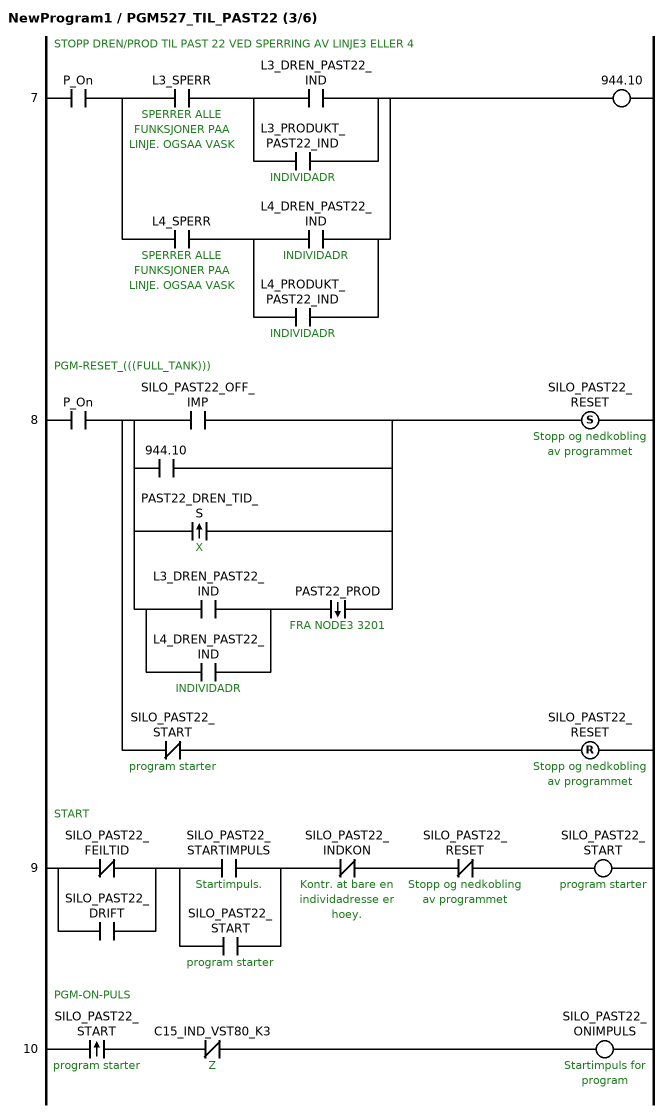
; rung 7: STOPP DREN/PROD TIL PAST 22 VED SPERRING AV LINJE3 ELLER 4
LD P_On
LD L3_SPERR  ; SPERRER ALLE FUNKSJONER PAA LINJE. OGSAA VASK
LD L3_DREN_PAST22_IND
OR L3_PRODUKT_PAST22_IND  ; INDIVIDADR
ANDLD
LD L4_SPERR  ; SPERRER ALLE FUNKSJONER PAA LINJE. OGSAA VASK
LD L4_DREN_PAST22_IND  ; INDIVIDADR
OR L4_PRODUKT_PAST22_IND  ; INDIVIDADR
ANDLD
ORLD
ANDLD
OUT 944.10
; rung 8: PGM-RESET_(((FULL_TANK)))
LD P_On
OUT TR0
LD SILO_PAST22_OFF_IMP
OR 944.10
@OR PAST22_DREN_TID_S  ; X
LD L3_DREN_PAST22_IND
OR L4_DREN_PAST22_IND  ; INDIVIDADR
%AND PAST22_PROD  ; FRA NODE3 3201
ORLD
ANDLD
SET SILO_PAST22_RESET  ; Stopp og nedkobling av programmet
LD TR0
ANDNOT SILO_PAST22_START  ; program starter
RSET SILO_PAST22_RESET  ; Stopp og nedkobling av programmet
; rung 9: START
LDNOT SILO_PAST22_FEILTID
OR SILO_PAST22_DRIFT
LD SILO_PAST22_STARTIMPULS  ; Startimpuls.
OR SILO_PAST22_START  ; program starter
ANDLD
ANDNOT SILO_PAST22_INDKON  ; Kontr. at bare en individadresse er hoey.
ANDNOT SILO_PAST22_RESET  ; Stopp og nedkobling av programmet
OUT SILO_PAST22_START  ; program starter
; rung 10: PGM-ON-PULS
@LD SILO_PAST22_START  ; program starter
ANDNOT C15_IND_VST80_K3  ; Z
OUT SILO_PAST22_ONIMPULS  ; Startimpuls for  program

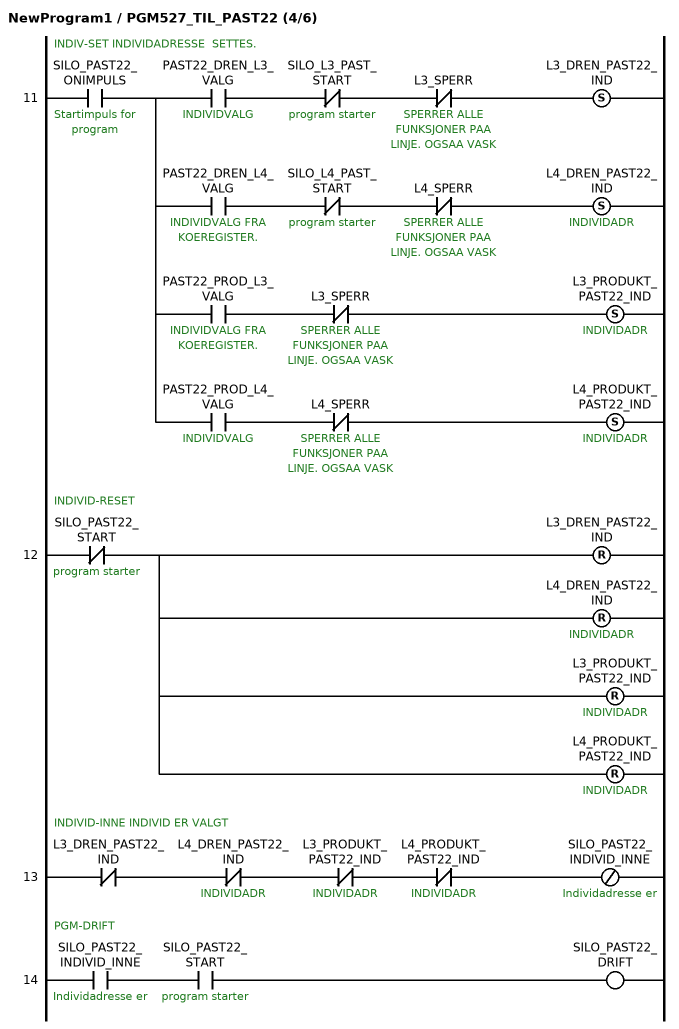
; rung 11: INDIV-SET INDIVIDADRESSE  SETTES.
LD SILO_PAST22_ONIMPULS  ; Startimpuls for  program
OUT TR0
AND PAST22_DREN_L3_VALG  ; INDIVIDVALG
ANDNOT SILO_L3_PAST_START  ; program starter
ANDNOT L3_SPERR  ; SPERRER ALLE FUNKSJONER PAA LINJE. OGSAA VASK
SET L3_DREN_PAST22_IND
LD TR0
AND PAST22_DREN_L4_VALG  ; INDIVIDVALG FRA KOEREGISTER.
ANDNOT SILO_L4_PAST_START  ; program starter
ANDNOT L4_SPERR  ; SPERRER ALLE FUNKSJONER PAA LINJE. OGSAA VASK
SET L4_DREN_PAST22_IND  ; INDIVIDADR
LD TR0
AND PAST22_PROD_L3_VALG  ; INDIVIDVALG FRA KOEREGISTER.
ANDNOT L3_SPERR  ; SPERRER ALLE FUNKSJONER PAA LINJE. OGSAA VASK
SET L3_PRODUKT_PAST22_IND  ; INDIVIDADR
LD TR0
AND PAST22_PROD_L4_VALG  ; INDIVIDVALG
ANDNOT L4_SPERR  ; SPERRER ALLE FUNKSJONER PAA LINJE. OGSAA VASK
SET L4_PRODUKT_PAST22_IND  ; INDIVIDADR
; rung 12: INDIVID-RESET
LDNOT SILO_PAST22_START  ; program starter
RSET L3_DREN_PAST22_IND
RSET L4_DREN_PAST22_IND  ; INDIVIDADR
RSET L3_PRODUKT_PAST22_IND  ; INDIVIDADR
RSET L4_PRODUKT_PAST22_IND  ; INDIVIDADR
; rung 13: INDIVID-INNE INDIVID ER VALGT
LDNOT L3_DREN_PAST22_IND
ANDNOT L4_DREN_PAST22_IND  ; INDIVIDADR
ANDNOT L3_PRODUKT_PAST22_IND  ; INDIVIDADR
ANDNOT L4_PRODUKT_PAST22_IND  ; INDIVIDADR
OUTNOT SILO_PAST22_INDIVID_INNE  ; Individadresse er
; rung 14: PGM-DRIFT
LD SILO_PAST22_INDIVID_INNE  ; Individadresse er
AND SILO_PAST22_START  ; program starter
OUT SILO_PAST22_DRIFT

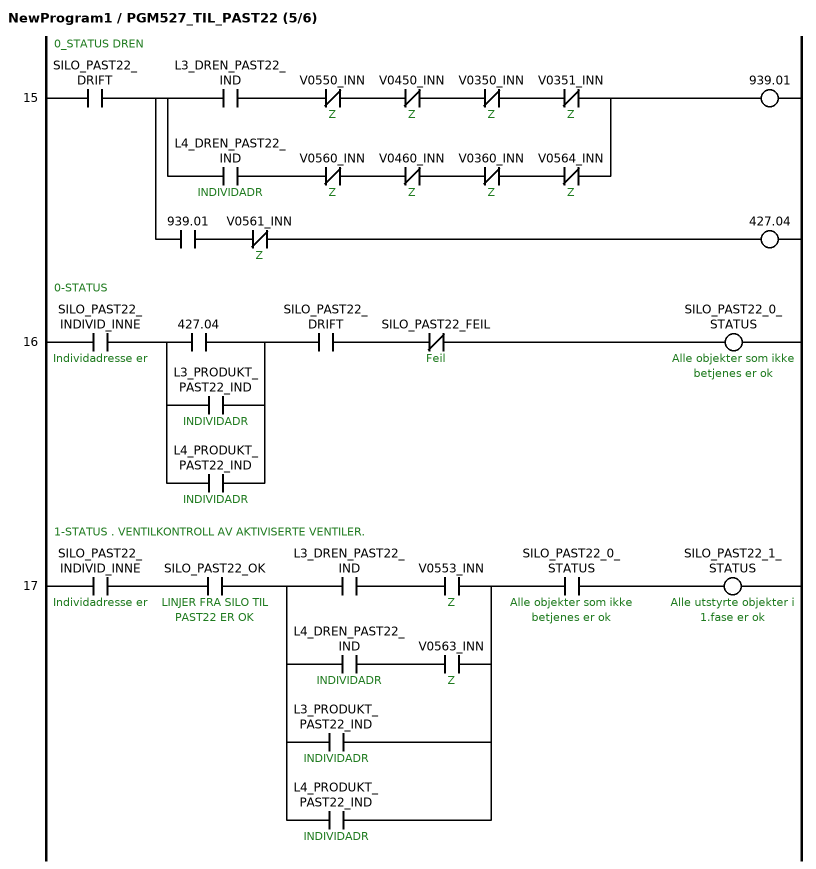
; rung 15: 0_STATUS DREN
LD SILO_PAST22_DRIFT
OUT TR0
LD L3_DREN_PAST22_IND
ANDNOT V0550_INN  ; Z
ANDNOT V0450_INN  ; Z
ANDNOT V0350_INN  ; Z
ANDNOT V0351_INN  ; Z
LD L4_DREN_PAST22_IND  ; INDIVIDADR
ANDNOT V0560_INN  ; Z
ANDNOT V0460_INN  ; Z
ANDNOT V0360_INN  ; Z
ANDNOT V0564_INN  ; Z
ORLD
ANDLD
OUT 939.01
LD TR0
AND 939.01
ANDNOT V0561_INN  ; Z
OUT 427.04
; rung 16: 0-STATUS
LD SILO_PAST22_INDIVID_INNE  ; Individadresse er
LD 427.04
OR L3_PRODUKT_PAST22_IND  ; INDIVIDADR
OR L4_PRODUKT_PAST22_IND  ; INDIVIDADR
ANDLD
AND SILO_PAST22_DRIFT
ANDNOT SILO_PAST22_FEIL  ; Feil
OUT SILO_PAST22_0_STATUS  ; Alle objekter som ikke betjenes er ok
; rung 17: 1-STATUS . VENTILKONTROLL AV AKTIVISERTE VENTILER.
LD SILO_PAST22_INDIVID_INNE  ; Individadresse er
AND SILO_PAST22_OK  ; LINJER FRA SILO TIL  PAST22 ER OK
LD L3_DREN_PAST22_IND
AND V0553_INN  ; Z
LD L4_DREN_PAST22_IND  ; INDIVIDADR
AND V0563_INN  ; Z
ORLD
OR L3_PRODUKT_PAST22_IND  ; INDIVIDADR
OR L4_PRODUKT_PAST22_IND  ; INDIVIDADR
ANDLD
AND SILO_PAST22_0_STATUS  ; Alle objekter som ikke betjenes er ok
OUT SILO_PAST22_1_STATUS  ; Alle utstyrte objekter i 1.fase er ok

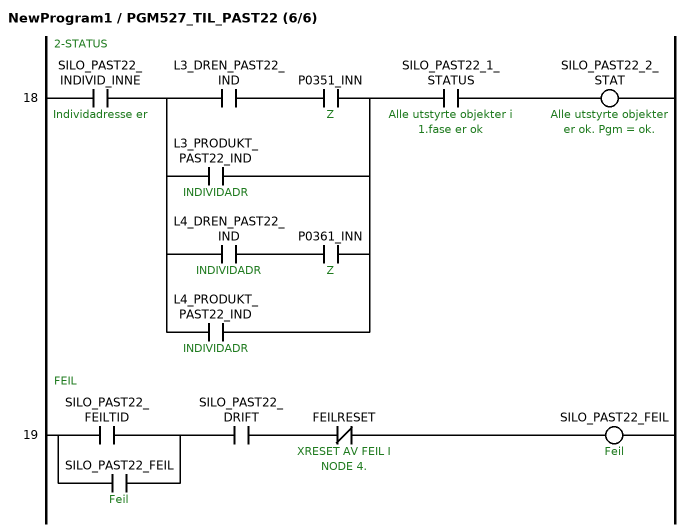
; rung 18: 2-STATUS
LD SILO_PAST22_INDIVID_INNE  ; Individadresse er
LD L3_DREN_PAST22_IND
AND P0351_INN  ; Z
OR L3_PRODUKT_PAST22_IND  ; INDIVIDADR
LD L4_DREN_PAST22_IND  ; INDIVIDADR
AND P0361_INN  ; Z
ORLD
OR L4_PRODUKT_PAST22_IND  ; INDIVIDADR
ANDLD
AND SILO_PAST22_1_STATUS  ; Alle utstyrte objekter i 1.fase er ok
OUT SILO_PAST22_2_STAT  ; Alle utstyrte objekter er ok. Pgm = ok.
; rung 19: FEIL
LD SILO_PAST22_FEILTID
OR SILO_PAST22_FEIL  ; Feil
AND SILO_PAST22_DRIFT
ANDNOT FEILRESET  ; XRESET AV FEIL I NODE 4.
OUT SILO_PAST22_FEIL  ; Feil

### Section L4_STATUS

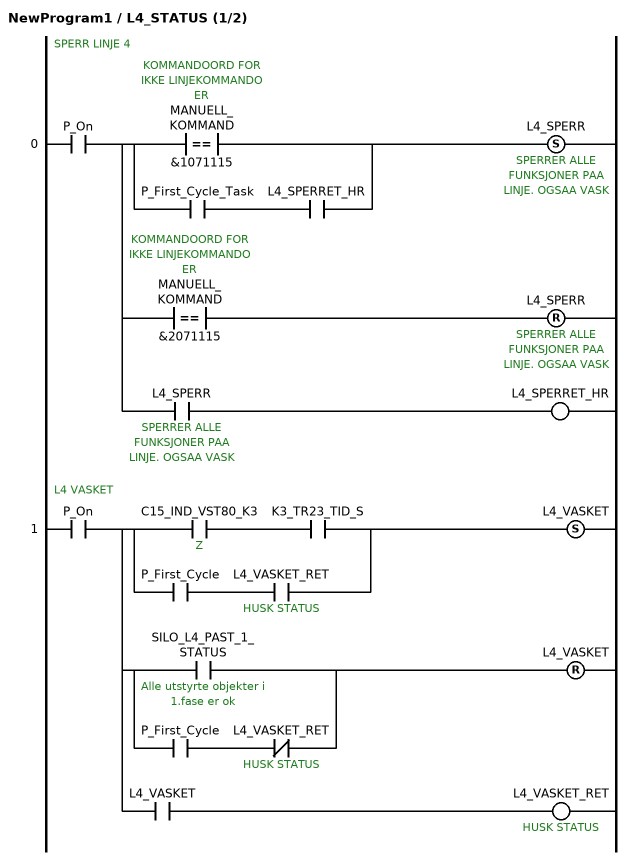
; rung 0: SPERR LINJE 4
LD P_On
OUT TR0
LD=L(301) MANUELL_KOMMAND &1071115  ; KOMMANDOORD FOR IKKE LINJEKOMMANDOER
LD P_First_Cycle_Task
AND L4_SPERRET_HR
ORLD
ANDLD
SET L4_SPERR  ; SPERRER ALLE FUNKSJONER PAA LINJE. OGSAA VASK
LD TR0
AND=L(301) MANUELL_KOMMAND &2071115  ; KOMMANDOORD FOR IKKE LINJEKOMMANDOER
RSET L4_SPERR  ; SPERRER ALLE FUNKSJONER PAA LINJE. OGSAA VASK
LD TR0
AND L4_SPERR  ; SPERRER ALLE FUNKSJONER PAA LINJE. OGSAA VASK
OUT L4_SPERRET_HR
; rung 1: L4 VASKET
LD P_On
OUT TR0
LD C15_IND_VST80_K3  ; Z
AND K3_TR23_TID_S
LD P_First_Cycle
AND L4_VASKET_RET  ; HUSK STATUS
ORLD
ANDLD
SET L4_VASKET
LD TR0
LD SILO_L4_PAST_1_STATUS  ; Alle utstyrte objekter i 1.fase er ok
LD P_First_Cycle
ANDNOT L4_VASKET_RET  ; HUSK STATUS
ORLD
ANDLD
RSET L4_VASKET
LD TR0
AND L4_VASKET
OUT L4_VASKET_RET  ; HUSK STATUS

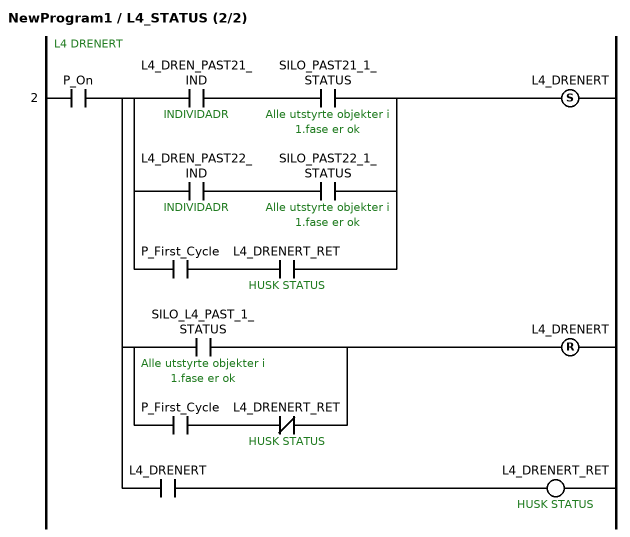
; rung 2: L4 DRENERT
LD P_On
OUT TR0
LD L4_DREN_PAST21_IND  ; INDIVIDADR
AND SILO_PAST21_1_STATUS  ; Alle utstyrte objekter i 1.fase er ok
LD L4_DREN_PAST22_IND  ; INDIVIDADR
AND SILO_PAST22_1_STATUS  ; Alle utstyrte objekter i 1.fase er ok
ORLD
LD P_First_Cycle
AND L4_DRENERT_RET  ; HUSK STATUS
ORLD
ANDLD
SET L4_DRENERT
LD TR0
LD SILO_L4_PAST_1_STATUS  ; Alle utstyrte objekter i 1.fase er ok
LD P_First_Cycle
ANDNOT L4_DRENERT_RET  ; HUSK STATUS
ORLD
ANDLD
RSET L4_DRENERT
LD TR0
AND L4_DRENERT
OUT L4_DRENERT_RET  ; HUSK STATUS

### Section PGM528_L3_L4_TIL_PAST23

